INTERFACE IF_TeilHolen

METHOD holenAnfordern
VAR_INPUT
END_VAR
END_METHOD

METHOD teilHolen : BOOL
VAR_INPUT
END_VAR
END_METHOD

END_INTERFACE

(* stored: Version 1.1.0.1, ProductVersion 3.1.4024.12
   Itf IF_TeilHolen: Id {613d4a21-8024-4d01-8b02-dd614f2582a8}
   Method holenAnfordern: Id {4924966c-4666-47de-accb-40619baf1922}
   Method teilHolen: Id {32ecd279-038d-45c5-9083-48ccc08ca6b5} *)
